FUNCTION TryConvert_LINT_TO_LREAL : BOOL
VAR_INPUT
	in : LINT;
	out : REFERENCE TO LREAL;
END_VAR

out := LINT_TO_LREAL(in);
TryConvert_LINT_TO_LREAL := TRUE;

END_FUNCTION

(* stored: Version 1.1.0.1, ProductVersion 3.1.4024.12
   POU TryConvert_LINT_TO_LREAL: Id {93a8b374-9c17-4fd2-b409-793baba9dbb4}, SpecialFunc None *)
